// TIA Portal V17 export
// export: Created 2025-06-26T06:49:19.7521022Z, ExportSetting WithDefaults, DisplayName Totally Integrated Automation Portal, DisplayVersion V17 Update 8, DisplayName TIA Portal Openness, DisplayVersion V17 Update 8, DisplayName TIA Portal Version Control Interface, DisplayVersion V17, DisplayName STEP 7 Professional, DisplayVersion V17 Update 8, DisplayName STEP 7 Safety, DisplayVersion V17 Update 6, DisplayName WinCC Advanced, DisplayVersion V17 Update 8
FUNCTION "isNotNaN" : Bool   // FC21, FBD
TITLE = isNotNaN
{ S7_Optimized_Access := 'TRUE' }
VERSION : 0.1
// Returns TRUE if a REAL is not NaN
// stored: AutoNumber true, IsIECCheckEnabled false, SetENOAutomatically false, UDAEnableTagReadback false
   VAR_INPUT
      In : Real;
   END_VAR
BEGIN

REGION Network 1
   // OK is a compiler builtin, but not available in SCL
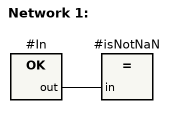
   // no SCL statement known for OK: written as a call
   #isNotNaN := OK(#In);
END_REGION
END_FUNCTION
